(* CoDeSys 2.3 export: START.EXP *)

(* POU start, ST *)
PROGRAM start
VAR

	test0 AT %QX0.0:BOOL;
END_VAR
test0 := 0;
END_PROGRAM
